FUNCTION_BLOCK PrinterMock IMPLEMENTS IPrinter
VAR_INPUT
END_VAR
VAR_OUTPUT
END_VAR
VAR
END_VAR

METHOD get_output : STRING(255)
VAR_INPUT
END_VAR
END_METHOD

{warning 'add method implementation'}
METHOD print
END_METHOD

END_FUNCTION_BLOCK

(* stored: Version 1.1.0.1, ProductVersion 3.1.4022.7
   POU PrinterMock: Id {d9744287-16f0-4a89-a520-2fb915872022}, SpecialFunc None
   Method get_output: Id {5cece63a-8a94-4427-ad4e-8cef92b0d800}
   Method print: Id {4f3bfdef-3848-4c83-8ac1-319bb95b1fee} *)
